FUNCTION_BLOCK FB_TEST
VAR_INPUT
	bVentil : BOOL;
END_VAR
VAR_OUTPUT
	bDoorc : BOOL;
	bDooro : BOOL;
END_VAR
VAR
END_VAR

IF bVentil := FALSE
	//animation.delay (500);
	bDooro := TRUE;
END_IF

IF bVentil := TRUE
	//animation.delay (500);
	bDoorc := FALSE;
END_IF

END_FUNCTION_BLOCK

(* stored: Version 1.1.0.1, ProductVersion 3.1.4024.15
   POU FB_TEST: Id {99a1af79-e974-4698-ab19-71e4457ded0e}, SpecialFunc None *)
